INTERFACE IPointerEnumerator EXTENDS IObject

// Shows curent collection element
PROPERTY ABSTRACT Current : PVOID
GET
END_GET
END_PROPERTY

// Moves Current pointer to next collection element
METHOD MoveNext : BOOL
END_METHOD

// Sets the enumerator to its initial position, which is before the first element in the collection
METHOD Reset
END_METHOD

END_INTERFACE

(* stored: Version 1.1.0.1
   Itf IPointerEnumerator: Id {cf549bf9-3271-4139-bc61-748e47b5395e}
   Property Current: Id {5a4a9f37-47f9-4ee9-8ee2-4a81c80e0ec8}
   Get Get: Id {9ee9bc47-7616-46c9-92bc-608f2f478cc6}
   Method MoveNext: Id {2bf714dd-2998-4a0a-b518-6aac977ac38f}
   Method Reset: Id {ff66a34c-30d7-455e-826d-90c20ab3efe1} *)
